# B&R Automation Studio project ASmodeling
Automation Studio 4.9

## Configuration Config1

CPU 4PP065.0571-P74, AutomationRuntime D4.52, Build 4.1.2, Safety 1.6, Vc V4.52.0

### Hardware
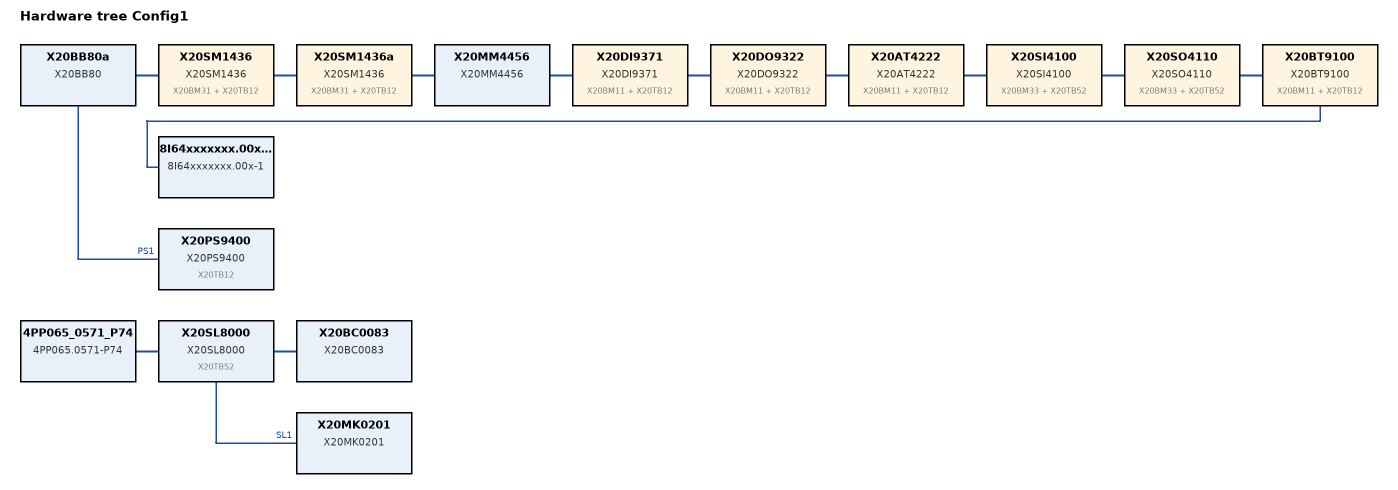
```
4PP065_0571_P74 : 4PP065.0571-P74 v1.1.2.0
  Connector IF4:
    DNAConfiguration = manual
  Connector IF5:
    ActivateDevice = 1
    Mode = Manual
    InternetAddress = 10.0.1.1
    SubnetMask = 255.255.255.0
  ConfigurationID = fdsagas_Config1
  Simulation = 1
  TimerDeviceType = EPLX2X
  TimerDevice = 4PP065_0571_P74.IF4
  TaskClassIdleTime = 2000
  Cyclic1Duration = 2000
  Cyclic1Tolerance = 0
  Cyclic1Output = 1
  FileDevice1
  FileDeviceName1 = USER
  FileDevicePath1 = USER_PATH
8I64xxxxxxx.00x-1 : 8I64xxxxxxx.00x-1 v2.1.1.0  [X2X1 -> X20BT9100.X2X1 [Cable Type=X2XCable, Length=10, Version=1.0.0.3]]
  FunctionModel = Standard
X20AT4222 : X20AT4222 v1.3.0.0  [SS1 -> X20TB12f.SS; SL -> X20BM11c.SL1]
X20BB80a : X20BB80 v1.0.2.0
X20BC0083 : X20BC0083 v2.11.1.0  [PLK1 -> X20SL8000.PLK2 (NodeNumber=2) [Cable Type=PowerlinkCable, Length=10, Version=1.0.0.3]; SL -> X20BB80a.SL1]
X20BM11a : X20BM11 v1.0.0.1  [X2X1 -> X20MM4456.X2X2]
X20BM11b : X20BM11 v1.0.0.1  [X2X1 -> X20BM11a.X2X2]
X20BM11c : X20BM11 v1.0.0.1  [X2X1 -> X20BM11b.X2X2]
X20BM11d : X20BM11 v1.0.0.1  [X2X1 -> X20BM33b.X2X2]
X20BM31a : X20BM31 v1.0.0.1  [X2X1 -> X20BB80a.IF1]
X20BM31b : X20BM31 v1.0.0.1  [X2X1 -> X20BM31a.X2X2]
X20BM33a : X20BM33 v1.0.0.6  [X2X1 -> X20BM11c.X2X2]
X20BM33b : X20BM33 v1.0.0.6  [X2X1 -> X20BM33a.X2X2]
X20BT9100 : X20BT9100 v1.1.0.0  [SS1 -> X20TB12g.SS; SL -> X20BM11d.SL1]
X20DI9371 : X20DI9371 v1.1.0.0  [SS1 -> X20TB12d.SS; SL -> X20BM11a.SL1]
X20DO9322 : X20DO9322 v1.3.0.0  [SS1 -> X20TB12e.SS; SL -> X20BM11b.SL1]
X20MK0201 : X20MK0201 v1.0.0.0  [SL -> X20SL8000.SL1]
X20MM4456 : X20MM4456 v1.4.0.0  [X2X1 -> X20BM31b.X2X2]
X20PS9400 : X20PS9400 v1.5.0.0  [SS1 -> X20TB12.SS; PS -> X20BB80a.PS1]
X20SI4100 : X20SI4100 v1.10.11.0  [SS1 -> X20TB52b.SS; SL -> X20BM33a.SL1]
X20SL8000 : X20SL8000 v1.6.5.2  [PLK1 -> 4PP065_0571_P74.IF4 (NodeNumber=1) [Cable Type=PowerlinkCable, Length=10, Version=1.0.0.3]; PLK2 -> X20BC0083.PLK1 (NodeNumber=1) [Cable Type=PowerlinkCable, Length=10, Version=1.0.0.3]; SS1 -> X20TB52.SS]
  SafeProject = SafeLOGIC-1
X20SM1436 : X20SM1436 v2.2.1.0  [SS1 -> X20TB12a.SS; SL -> X20BM31a.SL1]
  BothEndSwitchesAreNormallyOpen_r1 = on
  QuickStopIsNormallyOpen_r1 = on
X20SM1436a : X20SM1436 v2.2.1.0  [SS1 -> X20TB12c.SS; SL -> X20BM31b.SL1]
  BothEndSwitchesAreNormallyOpen_r1 = on
  QuickStopIsNormallyOpen_r1 = on
X20SO4110 : X20SO4110 v1.10.11.0  [SS1 -> X20TB52c.SS; SL -> X20BM33b.SL1]
  SafeModuleID = 3
X20TB12 : X20TB12 v1.0.0.0
X20TB12a : X20TB12 v1.0.0.0
X20TB12c : X20TB12 v1.0.0.0
X20TB12d : X20TB12 v1.0.0.0
X20TB12e : X20TB12 v1.0.0.0
X20TB12f : X20TB12 v1.0.0.0
X20TB12g : X20TB12 v1.0.0.0
X20TB52 : X20TB52 v1.0.0.2
X20TB52b : X20TB52 v1.0.0.2
X20TB52c : X20TB52 v1.0.0.2
```

## Logical view

### Library Logical/Libraries/Library (ANSIC)

#### Library.fun - Exported functions and function blocks
```iecst
{REDUND_ERROR} {REDUND_UNREPLICABLE} FUNCTION_BLOCK FB_integraotor (*TODO: Add your comment here*) (*$GROUP=User,$CAT=User,$GROUPICON=User.png,$CATICON=User.png*)
	VAR_INPUT
		in : {REDUND_UNREPLICABLE} REAL; (*вход интегрирующего звена*)
	END_VAR
	VAR_OUTPUT
		out : {REDUND_UNREPLICABLE} REAL; (*выход интегрирующего звена*)
	END_VAR
	VAR
		dt : {REDUND_UNREPLICABLE} REAL; (*шаг расчета [с]*)
		oldval : {REDUND_UNREPLICABLE} REAL; (*J*)
	END_VAR
END_FUNCTION_BLOCK

{REDUND_ERROR} FUNCTION_BLOCK FB_motor (*TODO: Add your comment here*) (*$GROUP=User,$CAT=User,$GROUPICON=User.png,$CATICON=User.png*)
	VAR_INPUT
		u : REAL; (*входное напряжение [В]*)
		Tm : REAL; (*частота вращения [об/мин]*)
	END_VAR
	VAR_OUTPUT
		w : REAL; (*интегратор *)
		phi : REAL; (*электромеханическая постоянная времени [с]*)
	END_VAR
	VAR
		ke : REAL; (*положение [рад]*)
		integraotor : FB_integraotor; (*постоянная ЭДС двигателя [В•мин/об]*)
		dt : REAL; (*шаг расчета [с]*)
	END_VAR
END_FUNCTION_BLOCK

FUNCTION_BLOCK FB_regulator
	VAR
		e : REAL; (*рассогласование между задающим воздействием и реальной скоростью вращения вала ДПТ [об/мин]*)
		u : REAL; (*напряжение, подаваемое на вход ДПТ [В]*)
		k_p : REAL; (*пропорциональный коэффициент регулятора*)
		k_i : REAL; (*интегральный коэффициент регулятора*)
		integrator : FB_integraotor; (*интегратор *)
		iyOld : REAL; (*хранение предыдущего значения схемы противонакопления*)
		max_abs_value : REAL; (*граница блока ограничения [В]*)
		dt : REAL; (*шаг расчета [с]*)
	END_VAR
END_FUNCTION_BLOCK

{REDUND_ERROR} {REDUND_UNREPLICABLE} FUNCTION_BLOCK FB_motor1 (*TODO: Add your comment here*) (*$GROUP=User,$CAT=User,$GROUPICON=User.png,$CATICON=User.png*)
	VAR_INPUT
		u : REAL; (*входное напряжение [В]*)
		Tm : REAL; (*частота вращения [об/мин]*)
	END_VAR
	VAR_OUTPUT
		w : REAL; (*интегратор *)
		phi : REAL; (*электромеханическая постоянная времени [с]*)
	END_VAR
	VAR
		ke : REAL; (*положение [рад]*)
		integraotor : FB_integraotor; (*постоянная ЭДС двигателя [В•мин/об]*)
		dt : REAL; (*шаг расчета [с]*)
	END_VAR
END_FUNCTION_BLOCK
```

#### FB_integraotor.c
```c
\
#include <bur/plctypes.h>
#ifdef __cplusplus
	extern "C"
	{
#endif
	#include "Library.h"
#ifdef __cplusplus
	};
#endif
/* TODO: Add your comment here */
void FB_integraotor(struct FB_integraotor* inst)
{

	inst->out = inst->oldval + ((inst->in) * inst->dt);
	inst->oldval = inst->out;
	/*TODO: Add your code here*/
}
```

#### FB_motor.c
```c
#include <bur/plctypes.h>
#ifdef __cplusplus
	extern "C"
	{
#endif
	#include "Library.h"
#ifdef __cplusplus
	};
#endif
/* TODO: Add your comment here */
void FB_motor(struct FB_motor* inst)
{
	REAL temp;
	temp = inst->u / inst->ke;
	temp = temp - inst->w;
	temp = temp * inst->dt / inst->Tm;
	inst->integraotor.in = temp;
	inst->integraotor.dt = inst->dt;
	FB_integraotor(&inst->integraotor);
	temp = inst->integraotor.out;
	inst->w = temp;
	temp = inst->w;
	inst->integraotor.in = temp;
	FB_integraotor(&inst->integraotor);
	inst->phi = inst->phi + temp;
	/*TODO: Add your code here*/
}
```

#### FB_regulator.c
```c
#include <bur/plctypes.h>
#ifdef __cplusplus
	extern "C"
	{
#endif
	#include "Library.h"
#ifdef __cplusplus
	};
#endif
/* TODO: Add your comment here */
void FB_regulator(struct FB_regulator* inst)
{

	REAL temp;
	temp = inst->e * inst->k_i * inst->dt;
	temp+=inst->iyOld;
	FB_integraotor(&inst->integrator);
	inst->integrator.in = temp;
	inst->integrator.dt = inst->dt;

	if (inst->e * inst->k_p > inst->max_abs_value)
	{
		temp = inst->integrator.out + inst->max_abs_value;
	}
	if (inst->e * inst->k_p < inst->max_abs_value)
	{
		temp = inst->integrator.out + inst->e * inst->k_p;
	}
	if (temp > inst->max_abs_value)
	{
		inst->u = inst->max_abs_value;
		inst->iyOld = temp - inst->max_abs_value;
	}
	else
	{
		inst->u = temp;
		inst->iyOld = 0;
	}

	/*TODO: Add your code here*/
}
```

#### FB_motor1.c
```c
#include <bur/plctypes.h>
#ifdef __cplusplus
	extern "C"
	{
#endif
	#include "Library.h"
#ifdef __cplusplus
	};
#endif
/* TODO: Add your comment here */
void FB_motor1(struct FB_motor1* inst)
{
	REAL temp;
	temp = inst->u / inst->ke;
	temp = temp - inst->w;
	temp = temp * inst->dt / inst->Tm;
	inst->integraotor.in = temp;
	inst->integraotor.dt = inst->dt;
	FB_integraotor(&inst->integraotor);
	temp = inst->integraotor.out;
	inst->w = temp;
	temp = inst->w;
	inst->integraotor.in = temp;
	FB_integraotor(&inst->integraotor);
	inst->phi = inst->phi + temp;
	/*TODO: Add your code here*/
}
```

### Program Logical/Program

#### Variables.var
```iecst
VAR
	fb_motor : FB_motor;
	Speed : REAL;
	fb_reg : FB_regulator;
	timecount : REAL;
	Enable : BOOL;
	t : REAL;
	ResW : REAL;
	ResPhi : REAL;
	fb_motor1 : FB_motor1;
END_VAR
```

#### Main.c
```c
#include <bur/plctypes.h>

#ifdef _DEFAULT_INCLUDES
	#include <AsDefault.h>
#endif

void _INIT ProgramInit(void)
{
	timecount = 0;

	t = 0;
	fb_motor.dt = 0.1;
	fb_motor.Tm = 0.1;
	fb_motor.ke = 1;

	fb_motor1.dt = 0.1;
	fb_motor1.Tm = 0.1;
	fb_motor1.ke = 1;

	fb_reg.dt = 0.001;
	fb_reg.e = 10;
	fb_reg.k_i = 1;
	fb_reg.k_p = 10;
	fb_reg.max_abs_value = 300;

}

void _CYCLIC ProgramCyclic(void)
{
	if (Enable == 1)
	{
		Speed = 100;
	}
	if (Enable == 0)
	{
		Speed = 0;
	}
	t = t + 0.1;
	timecount+=0.1;
	fb_reg.e = Speed - fb_motor.w;
	FB_regulator(&fb_reg);
	fb_motor.u = fb_reg.u;
	FB_motor(&fb_motor);
	ResW = fb_motor.w;
	ResPhi = fb_motor.phi;
	FB_motor1(&fb_motor1);
	fb_motor1.u = Speed - fb_motor1.w;

	if ((timecount>=5)&&(timecount<10)){
		Enable = 1;
	}
	if (timecount>=10){
		Enable = 0;

	}
	if (timecount>=15){
		timecount = 0;
		Enable = 1;\
	}
}

void _EXIT ProgramExit(void)
{

}
```

Listed in the project but not available here: Logical/Libraries/Library/Types.typ, Logical/Libraries/Library/Constants.var
